Staubli VAL3: saveData.dtx

public FrameItem fFrameItem[11]
  [0]
    frame fFrame = {fatherId=world[0]}
    pointRx pO = {fatherId=world[0]}
    pointRx pX = {fatherId=world[0]}
    pointRx pY = {fatherId=world[0]}
    string sName = "World"
  [1]
    frame fFrame = {fatherId=world[0]}
    pointRx pO = {fatherId=world[0]}
    pointRx pX = {fatherId=world[0]}
    pointRx pY = {fatherId=world[0]}
    string sName
  [2]
    frame fFrame = {fatherId=world[0]}
    pointRx pO = {fatherId=world[0]}
    pointRx pX = {fatherId=world[0]}
    pointRx pY = {fatherId=world[0]}
    string sName
  [3]
    frame fFrame = {fatherId=world[0]}
    pointRx pO = {fatherId=world[0]}
    pointRx pX = {fatherId=world[0]}
    pointRx pY = {fatherId=world[0]}
    string sName
  [4]
    frame fFrame = {fatherId=world[0]}
    pointRx pO = {fatherId=world[0]}
    pointRx pX = {fatherId=world[0]}
    pointRx pY = {fatherId=world[0]}
    string sName
  [5]
    frame fFrame = {fatherId=world[0]}
    pointRx pO = {fatherId=world[0]}
    pointRx pX = {fatherId=world[0]}
    pointRx pY = {fatherId=world[0]}
    string sName
  [6]
    frame fFrame = {fatherId=world[0]}
    pointRx pO = {fatherId=world[0]}
    pointRx pX = {fatherId=world[0]}
    pointRx pY = {fatherId=world[0]}
    string sName
  [7]
    frame fFrame = {fatherId=world[0]}
    pointRx pO = {fatherId=world[0]}
    pointRx pX = {fatherId=world[0]}
    pointRx pY = {fatherId=world[0]}
    string sName
  [8]
    frame fFrame = {fatherId=world[0]}
    pointRx pO = {fatherId=world[0]}
    pointRx pX = {fatherId=world[0]}
    pointRx pY = {fatherId=world[0]}
    string sName
  [9]
    frame fFrame = {fatherId=world[0]}
    pointRx pO = {fatherId=world[0]}
    pointRx pX = {fatherId=world[0]}
    pointRx pY = {fatherId=world[0]}
    string sName
  [10]
    frame fFrame = {fatherId=world[0]}
    pointRx pO = {fatherId=world[0]}
    pointRx pX = {fatherId=world[0]}
    pointRx pY = {fatherId=world[0]}
    string sName
public Instruction iInstruction{}
  [CALL]
    bool bIsTraj
    bool bUseOnPoint
    num nIndex
    string sID = "CALL"
    string sPath = "instruction/CALL"
  [DELAY]
    bool bIsTraj
    bool bUseOnPoint
    num nIndex = 1
    string sID = "DELAY"
    string sPath = "instruction/DELAY"
  [HOME]
    bool bIsTraj = true
    bool bUseOnPoint
    num nIndex = 10
    string sID = "HOME"
    string sPath = "trajectory/HOME"
  [IF]
    bool bIsTraj
    bool bUseOnPoint
    num nIndex = 2
    string sID = "IF"
    string sPath = "instruction/IF"
  [IN]
    bool bIsTraj
    bool bUseOnPoint
    num nIndex = 6
    string sID = "IN"
    string sPath = "instruction/inputOutput/IN"
  [JPOINT]
    bool bIsTraj = true
    bool bUseOnPoint
    num nIndex = 11
    string sID = "JPOINT"
    string sPath = "trajectory/JPOINT"
  [NUM]
    bool bIsTraj
    bool bUseOnPoint
    num nIndex = 7
    string sID = "NUM"
    string sPath = "instruction/inputOutput/NUM"
  [OUT]
    bool bIsTraj
    bool bUseOnPoint
    num nIndex = 8
    string sID = "OUT"
    string sPath = "instruction/inputOutput/OUT"
  [PALLET]
    bool bIsTraj = true
    bool bUseOnPoint
    num nIndex = 12
    string sID = "PALLET"
    string sPath = "trajectory/PALLET"
  [POINT]
    bool bIsTraj = true
    bool bUseOnPoint
    num nIndex = 13
    string sID = "POINT"
    string sPath = "trajectory/POINT"
  [PROG]
    bool bIsTraj
    bool bUseOnPoint
    num nIndex = 3
    string sID = "PROG"
    string sPath = "instruction/PROG"
  [PULSE]
    bool bIsTraj
    bool bUseOnPoint
    num nIndex = 4
    string sID = "PULSE"
    string sPath = "instruction/PULSE"
  [SUB]
    bool bIsTraj
    bool bUseOnPoint
    num nIndex = 5
    string sID = "SUB"
    string sPath = "instruction/SUB"
  [TRAJ]
    bool bIsTraj = true
    bool bUseOnPoint
    num nIndex = 14
    string sID = "TRAJ"
    string sPath = "trajectory/TRAJ"
  [WAIT]
    bool bIsTraj
    bool bUseOnPoint
    num nIndex = 9
    string sID = "WAIT"
    string sPath = "instruction/inputOutput/WAIT"
public ToolItem tData[11]
  [0]
    InstrItem iActionOFF[3]
      [0]
        string sData
        string sType
      [1]
        string sData
        string sType
      [2]
        string sData
        string sType
    InstrItem iActionON[3]
      [0]
        string sData
        string sType
      [1]
        string sData
        string sType
      [2]
        string sData
        string sType
    string name = "flange"
    tool tcp = {fatherId=flange[0], ioLink=valve1}
  [1]
    InstrItem iActionOFF[3]
      [0]
        string sData
        string sType
      [1]
        string sData
        string sType
      [2]
        string sData
        string sType
    InstrItem iActionON[3]
      [0]
        string sData
        string sType
      [1]
        string sData
        string sType
      [2]
        string sData
        string sType
    string name
    tool tcp = {fatherId=flange[0], ioLink=valve1}
  [2]
    InstrItem iActionOFF[3]
      [0]
        string sData
        string sType
      [1]
        string sData
        string sType
      [2]
        string sData
        string sType
    InstrItem iActionON[3]
      [0]
        string sData
        string sType
      [1]
        string sData
        string sType
      [2]
        string sData
        string sType
    string name
    tool tcp = {fatherId=flange[0], ioLink=valve1}
  [3]
    InstrItem iActionOFF[3]
      [0]
        string sData
        string sType
      [1]
        string sData
        string sType
      [2]
        string sData
        string sType
    InstrItem iActionON[3]
      [0]
        string sData
        string sType
      [1]
        string sData
        string sType
      [2]
        string sData
        string sType
    string name
    tool tcp = {fatherId=flange[0], ioLink=valve1}
  [4]
    InstrItem iActionOFF[3]
      [0]
        string sData
        string sType
      [1]
        string sData
        string sType
      [2]
        string sData
        string sType
    InstrItem iActionON[3]
      [0]
        string sData
        string sType
      [1]
        string sData
        string sType
      [2]
        string sData
        string sType
    string name
    tool tcp = {fatherId=flange[0], ioLink=valve1}
  [5]
    InstrItem iActionOFF[3]
      [0]
        string sData
        string sType
      [1]
        string sData
        string sType
      [2]
        string sData
        string sType
    InstrItem iActionON[3]
      [0]
        string sData
        string sType
      [1]
        string sData
        string sType
      [2]
        string sData
        string sType
    string name
    tool tcp = {fatherId=flange[0], ioLink=valve1}
  [6]
    InstrItem iActionOFF[3]
      [0]
        string sData
        string sType
      [1]
        string sData
        string sType
      [2]
        string sData
        string sType
    InstrItem iActionON[3]
      [0]
        string sData
        string sType
      [1]
        string sData
        string sType
      [2]
        string sData
        string sType
    string name
    tool tcp = {fatherId=flange[0], ioLink=valve1}
  [7]
    InstrItem iActionOFF[3]
      [0]
        string sData
        string sType
      [1]
        string sData
        string sType
      [2]
        string sData
        string sType
    InstrItem iActionON[3]
      [0]
        string sData
        string sType
      [1]
        string sData
        string sType
      [2]
        string sData
        string sType
    string name
    tool tcp = {fatherId=flange[0], ioLink=valve1}
  [8]
    InstrItem iActionOFF[3]
      [0]
        string sData
        string sType
      [1]
        string sData
        string sType
      [2]
        string sData
        string sType
    InstrItem iActionON[3]
      [0]
        string sData
        string sType
      [1]
        string sData
        string sType
      [2]
        string sData
        string sType
    string name
    tool tcp = {fatherId=flange[0], ioLink=valve1}
  [9]
    InstrItem iActionOFF[3]
      [0]
        string sData
        string sType
      [1]
        string sData
        string sType
      [2]
        string sData
        string sType
    InstrItem iActionON[3]
      [0]
        string sData
        string sType
      [1]
        string sData
        string sType
      [2]
        string sData
        string sType
    string name
    tool tcp = {fatherId=flange[0], ioLink=valve1}
  [10]
    InstrItem iActionOFF[3]
      [0]
        string sData
        string sType
      [1]
        string sData
        string sType
      [2]
        string sData
        string sType
    InstrItem iActionON[3]
      [0]
        string sData
        string sType
      [1]
        string sData
        string sType
      [2]
        string sData
        string sType
    string name
    tool tcp = {fatherId=flange[0], ioLink=valve1}
public bool bChangeIO
public bool bCheck
public bool bDebug
public bool bInitAll
public bool bModbus
public bool bMultiSession
public bool bNoUseHome
public bool bPlc
public bool bPlcEnable
public bool bReloadList
public bool bShowItem
public bool bStopToPowerOff
public bool bToReload
public bool bUseBlendAction = true
public bool bUseHomeConfig
public bool bUseHomeScanner = true
public frame fAdjust = {fatherId=world[0]}
public frame fNewWorld[2]
  [0] = {fatherId=world[0]}
  [1] = {fatherId=world[0]}
public num mode = 2
public num nFrameActive
public num nFrameTool
public num nIndexTool
public num nRadiusHome = 400
public num nRound = 40
public num nSpeed = 100
public num nTimeDialog = -5
public num nTimeOut = -10
public pointRx rif2 = {fatherId=world[0]}
public string language = "chinese"
public string passwd[3]
  [0] = "programmer"
  [1] = "integrator"
  [2] = "toneage"
public string sInEnd
public string sInHome
public string sInStart
public string sInStop
public string sInstr[15]
  [0] = "CALL"
  [1] = "DELAY"
  [2] = "IF"
  [3] = "PROG"
  [4] = "PULSE"
  [5] = "SUB"
  [6] = "IN"
  [7] = "NUM"
  [8] = "OUT"
  [9] = "WAIT"
  [10] = "HOME"
  [11] = "JPOINT"
  [12] = "PALLET"
  [13] = "POINT"
  [14] = "TRAJ"
public string sInstrOnPoint[15]
  [0] = "CALL"
  [1] = "DELAY"
  [4] = "PULSE"
  [5] = "SUB"
  [6] = "IN"
  [7] = "NUM"
  [8] = "OUT"
  [9] = "WAIT"
public string sOutEnd
public string sOutHome
public string sOutStart
public string sOutStop
public string sPageLoad[17]
  [0] = "goHome/page_home_set"
  [1] = "instruction/PROG/page_instr"
  [2] = "instruction/PROG/page_program"
  [3] = "instruction/PROG/page_viewInstr"
  [4] = "instruction/inputOutput/page_inOut"
  [5] = "kernel/page/advance"
  [6] = "kernel/page/frame"
  [7] = "kernel/page/home"
  [8] = "kernel/page/processList"
  [9] = "kernel/page/production"
  [10] = "kernel/page/tool"
  [11] = "trajectory/PALLET/page_pallet"
  [12] = "trajectory/PALLET/page_viewPallet"
  [13] = "trajectory/page_editTraj"
  [14] = "trajectory/page_simulation"
  [15] = "trajectory/page_trajectory"
  [16] = "trajectory/page_viewTraj"
public string sPathPList = "Disk://session/default/saveCycle/"
public string sPathProg = "Disk://session/default/saveProg/"
public string sPathTraj = "Disk://session/default/saveTraj/"
public string sProgFilter
public string sProgType[3]
  [0] = "PROG"
  [1] = "SUB"
  [2] = "SERVICE"
public string sProgTypeUsing = "PROG"
public string sSession = "default"
public string sString
public string sTrajFilter
public string sTrajType[5]
  [0] = "HOME"
  [1] = "JPOINT"
  [2] = "PALLET"
  [3] = "POINT"
  [4] = "TRAJ"
public string sTrajTypeUsing = "TRAJ"
public tool tTool = {fatherId=flange[0], ioLink=valve1}
